Universal Robots PolyScope program: cable_extend_v3.urp

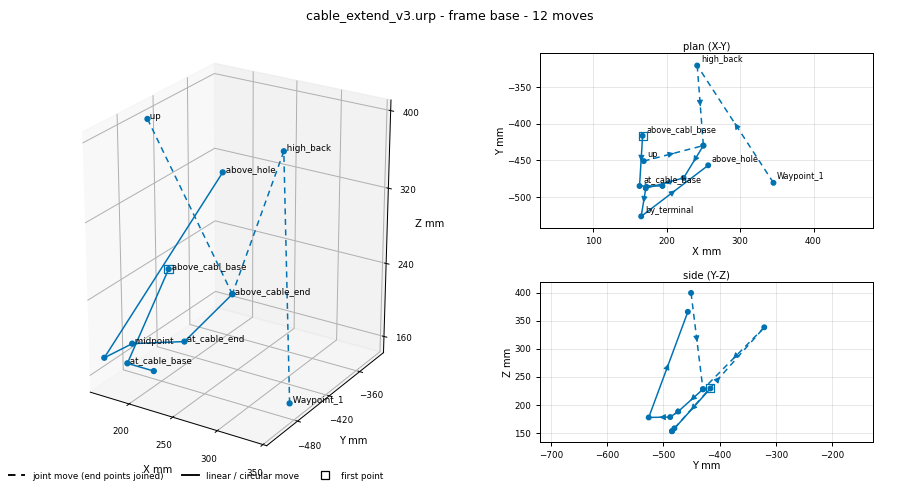
[picture p0: tool path of cable_extend_v3.urp in frame base, 12 of 14 moves have a stored position in this frame; points joined in program order, loops and branches not executed]
Program cable_extend_v3 (installation=default directory=/programs/wrs2020 createdIn=5.6.0.90886 lastSavedIn=5.9.1.1031110 robotSerialNumber=20205500180)
Calibrated DH parameters: a=[0, -0.425, -0.3922, 0, 0, 0]; d=[0.1625, 0, 0, 0.1333, 0.0997, 0.0996]; alpha=[1.570796, 0, 0, 1.570796, -1.570796, 0]; deltaTheta=[0, 0, 0, 0, 0, 0]
Robot Program (runOnlyOnce=true)
  URCap Gripper (Robotiq_Grippers, Robotiq Inc.) dataModel(position=71.76470588235294, force=0.0, speed=0.0, positionInDouble=71.76470588235294, forceInDouble=0.0, speedInDouble=0.0, slaveIds=[9], blocking=true)
  MoveL speed 250 mm/s, acceleration 1200 mm/s^2 (useActiveTCP=false) tcp=gripper_140_tip; feature=Base
    Waypoint above_cabl_base: TCP in base x=167.249 y=-416.393 z=229.475 mm, rx=1.8342 ry=-1.8019 rz=0.7367 rad; joints [94.618, -123.285, 140.281, -148.378, -89.759, -86.278] deg; TCP offset x=0 y=0 z=220 mm, rx=0 ry=0 rz=0 rad
    Waypoint at_cable_base: motionParameters(jointSpeed=1.047198 jointAcceleration=1.396263 cartesianSpeed=0.08 cartesianAcceleration=0.2); TCP in base x=163.077 y=-484.759 z=153.469 mm, rx=1.7934 ry=-1.8045 rz=0.6719 rad; joints [96.664, -101.667, 141.389, -170.745, -94.78, -84.635] deg
  URCap Gripper (Robotiq_Grippers, Robotiq Inc.) dataModel(position=84.31372549019608, force=0.0, speed=0.0, positionInDouble=84.31372549019608, forceInDouble=0.0, speedInDouble=0.0, slaveIds=[9], blocking=true)
  MoveL speed 250 mm/s, acceleration 1200 mm/s^2 (useActiveTCP=false) tcp=gripper_140_tip; feature=Base
    Waypoint wait_for_bbot: TCP in base x=194.304 y=-484.759 z=153.469 mm, rx=1.7934 ry=-1.8045 rz=0.6719 rad; joints [102.534, -98.816, 139.119, -170.778, -98.624, -80.153] deg
    Popup Message (haltProgram=false message=wait for b_bot to grasp cable. press enter to move together inputType=Text)
    Waypoint past_cable (Relative): motionParameters(jointSpeed=1.047198 jointAcceleration=1.396263 cartesianSpeed=0.01 cartesianAcceleration=1.2); relativeFromPosition TCP in base x=194.301 y=-484.746 z=153.444 mm, rx=1.7934 ry=-1.8045 rz=0.6718 rad; joints [102.533, -98.816, 139.121, -170.778, -98.622, -80.156] deg; TCP in base x=312.372 y=-484.763 z=153.441 mm, rx=1.7934 ry=-1.8046 rz=0.6719 rad; joints [120.436, -87.786, 128.042, -167.073, -109.898, -65.729] deg
    Waypoint Waypoint_1: TCP in base x=345.455 y=-480.429 z=158.653 mm, rx=1.9498 ry=-1.7894 rz=0.9532 rad; joints [113.534, -90.322, 133.097, -176.368, -91.379, -71.766] deg
  URCap Gripper (Robotiq_Grippers, Robotiq Inc.) dataModel(position=48.627450980392155, force=0.0, speed=100.0, positionInDouble=48.627450980392155, forceInDouble=0.0, speedInDouble=100.0, slaveIds=[9], blocking=true)
  MoveJ speed 60 deg/s, acceleration 80 deg/s^2 (useActiveTCP=false) tcp=gripper_140_tip; feature=Base
    Waypoint high_back: TCP in base x=241.615 y=-320.675 z=338.164 mm, rx=1.8342 ry=-1.8019 rz=0.7367 rad; joints [121.808, -127.577, 125.129, -125.645, -107.362, -65.273] deg
    Popup Message (haltProgram=false message=wait for b_bot to prepare cable. press enter to pick it inputType=Text)
    Waypoint above_cable_end: TCP in base x=250.005 y=-429.691 z=228.034 mm, rx=1.8342 ry=-1.802 rz=0.7366 rad; joints [112.09, -109.888, 133.785, -154.034, -101.413, -73.108] deg
  MoveL speed 250 mm/s, acceleration 1200 mm/s^2 (useActiveTCP=false) tcp=gripper_140_tip; feature=Base
    Waypoint at_cable_end: TCP in base x=223.11 y=-473.727 z=188.43 mm, rx=1.8342 ry=-1.8018 rz=0.7367 rad; joints [104.517, -103.353, 136.346, -164.041, -96.479, -78.931] deg
  URCap Gripper (Robotiq_Grippers, Robotiq Inc.) dataModel(position=100.0, force=100.0, speed=0.0, positionInDouble=100.0, forceInDouble=100.0, speedInDouble=0.0, slaveIds=[9], blocking=true)
  Popup Message (haltProgram=false message=press enter, then the robot will move to insert inputType=Text)
  MoveL speed 250 mm/s, acceleration 1200 mm/s^2 (useActiveTCP=false) tcp=gripper_140_tip; feature=Base
    Waypoint midpoint: TCP in base x=171.576 y=-487.871 z=178.568 mm, rx=1.6615 ry=-1.6465 rz=0.2212 rad; joints [116.588, -90.999, 128.222, -156.033, -128.334, -74.138] deg
    Waypoint by_terminal: TCP in base x=165.326 y=-526.084 z=177.926 mm, rx=1.7721 ry=-1.8956 rz=-0.0734 rad; joints [110.139, -84.302, 107.175, -123.092, -119.879, -68.738] deg
  MoveL speed 250 mm/s, acceleration 1200 mm/s^2 (useActiveTCP=false) tcp=TCP; feature=Base
    Waypoint above_hole: TCP in base x=256.585 y=-456.57 z=365.647 mm, rx=1.7722 ry=-1.8956 rz=-0.0734 rad; joints [110.141, -84.302, 107.175, -123.094, -119.877, -68.738] deg
    Popup Message (haltProgram=false message=press enter, then the robot will move to insert inputType=Text)
    Waypoint down (Relative): motionParameters(jointSpeed=1.047198 jointAcceleration=1.396263 cartesianSpeed=0.01 cartesianAcceleration=0.5); relativeFromPosition TCP in base x=169.213 y=-448.693 z=384.09 mm, rx=-0.0649 ry=3.0862 rz=-0.3319 rad; joints [94.252, -94.092, 112.857, -121.052, -88.362, 2.054] deg; TCP in base x=170.384 y=-459.976 z=363.444 mm, rx=-0.0649 ry=3.0862 rz=-0.3318 rad; joints [94.289, -91.461, 113.589, -124.413, -88.369, 2.104] deg
  URCap Gripper (Robotiq_Grippers, Robotiq Inc.) dataModel(position=78.43137254901961, force=0.0, speed=0.0, positionInDouble=78.43137254901961, forceInDouble=0.0, speedInDouble=0.0, slaveIds=[9], blocking=true)
  MoveJ speed 60 deg/s, acceleration 80 deg/s^2 (useActiveTCP=false) tcp=TCP; feature=Base
    Waypoint up: TCP in base x=168.816 y=-450.828 z=399.236 mm, rx=-0.0649 ry=3.0862 rz=-0.332 rad; joints [94.182, -94.491, 110.905, -118.704, -88.349, 1.979] deg
  MoveJ speed 60 deg/s, acceleration 80 deg/s^2 (useActiveTCP=false) tcp=gripper_140_tip; feature=Base
    Waypoint above_cable_end: TCP in base x=250.005 y=-429.691 z=228.034 mm, rx=1.8342 ry=-1.802 rz=0.7366 rad; joints [112.09, -109.888, 133.785, -154.034, -101.413, -73.108] deg; TCP offset x=0 y=0 z=220 mm, rx=0 ry=0 rz=0 rad
